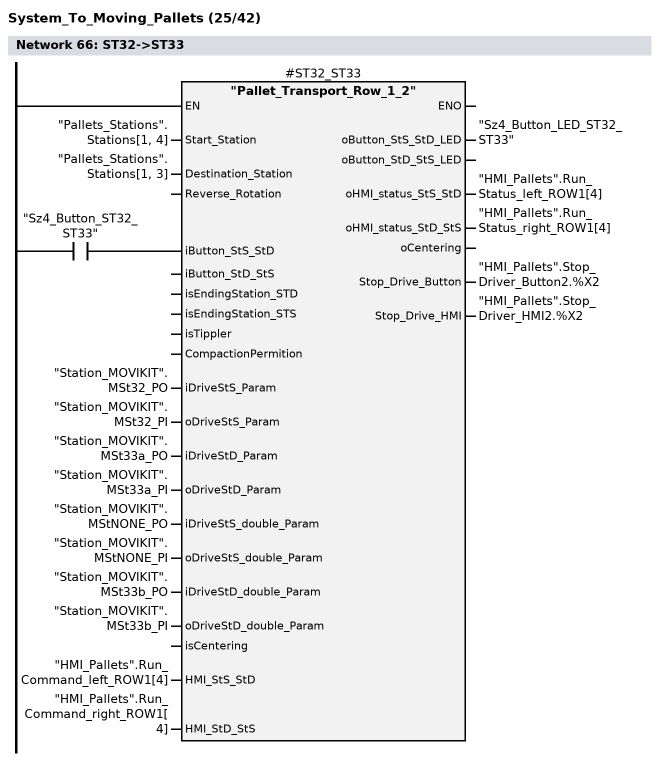
   RUNG wire#powerrail
      #ST32_ST33(iButton_StS_StD := wire#w1, Start_Station := "Pallets_Stations".Stations[1, 4], Destination_Station := "Pallets_Stations".Stations[1, 3], Reverse_Rotation :=, iButton_StD_StS :=, isEndingStation_STD :=, isEndingStation_STS :=, isTippler :=, CompactionPermition :=, iDriveStS_Param := "Station_MOVIKIT".MSt32_PO, oDriveStS_Param := "Station_MOVIKIT".MSt32_PI, iDriveStD_Param := "Station_MOVIKIT".MSt33a_PO, oDriveStD_Param := "Station_MOVIKIT".MSt33a_PI, iDriveStS_double_Param := "Station_MOVIKIT".MStNONE_PO, oDriveStS_double_Param := "Station_MOVIKIT".MStNONE_PI, iDriveStD_double_Param := "Station_MOVIKIT".MSt33b_PO, oDriveStD_double_Param := "Station_MOVIKIT".MSt33b_PI, isCentering :=, HMI_StS_StD := "HMI_Pallets".Run_Command_left_ROW1[4], HMI_StD_StS := "HMI_Pallets".Run_Command_right_ROW1[4], oButton_StS_StD_LED => "Sz4_Button_LED_ST32_ST33", oButton_StD_StS_LED =>, oHMI_status_StS_StD => "HMI_Pallets".Run_Status_left_ROW1[4], oHMI_status_StD_StS => "HMI_Pallets".Run_Status_right_ROW1[4], oCentering =>, Stop_Drive_Button => "HMI_Pallets".Stop_Driver_Button2.%X2, Stop_Drive_HMI => "HMI_Pallets".Stop_Driver_HMI2.%X2)
   END_RUNG
   RUNG wire#powerrail
      Contact( "Sz4_Button_ST32_ST33" )
   END_RUNG wire#w1
   // the same network as SCL:
   #ST32_ST33(Start_Station := "Pallets_Stations".Stations[1, 4],   // "Pallet_Transport_Row_1_2"
              Destination_Station := "Pallets_Stations".Stations[1, 3],
              iButton_StS_StD := "Sz4_Button_ST32_ST33",
              iDriveStS_Param := "Station_MOVIKIT".MSt32_PO,
              oDriveStS_Param := "Station_MOVIKIT".MSt32_PI,
              iDriveStD_Param := "Station_MOVIKIT".MSt33a_PO,
              oDriveStD_Param := "Station_MOVIKIT".MSt33a_PI,
              iDriveStS_double_Param := "Station_MOVIKIT".MStNONE_PO,
              oDriveStS_double_Param := "Station_MOVIKIT".MStNONE_PI,
              iDriveStD_double_Param := "Station_MOVIKIT".MSt33b_PO,
              oDriveStD_double_Param := "Station_MOVIKIT".MSt33b_PI,
              HMI_StS_StD := "HMI_Pallets".Run_Command_left_ROW1[4],
              HMI_StD_StS := "HMI_Pallets".Run_Command_right_ROW1[4],
              oButton_StS_StD_LED => "Sz4_Button_LED_ST32_ST33",
              oHMI_status_StS_StD => "HMI_Pallets".Run_Status_left_ROW1[4],
              oHMI_status_StD_StS => "HMI_Pallets".Run_Status_right_ROW1[4],
              Stop_Drive_Button => "HMI_Pallets".Stop_Driver_Button2.%X2,
              Stop_Drive_HMI => "HMI_Pallets".Stop_Driver_HMI2.%X2);
END_REGION

REGION Network 67: ST31->ST32
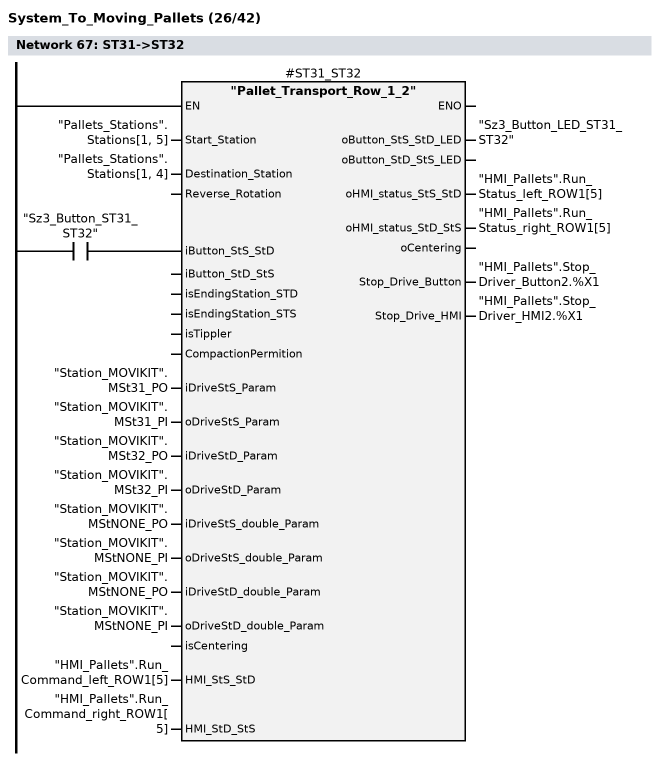
   RUNG wire#powerrail
      #ST31_ST32(iButton_StS_StD := wire#w1, Start_Station := "Pallets_Stations".Stations[1, 5], Destination_Station := "Pallets_Stations".Stations[1, 4], Reverse_Rotation :=, iButton_StD_StS :=, isEndingStation_STD :=, isEndingStation_STS :=, isTippler :=, CompactionPermition :=, iDriveStS_Param := "Station_MOVIKIT".MSt31_PO, oDriveStS_Param := "Station_MOVIKIT".MSt31_PI, iDriveStD_Param := "Station_MOVIKIT".MSt32_PO, oDriveStD_Param := "Station_MOVIKIT".MSt32_PI, iDriveStS_double_Param := "Station_MOVIKIT".MStNONE_PO, oDriveStS_double_Param := "Station_MOVIKIT".MStNONE_PI, iDriveStD_double_Param := "Station_MOVIKIT".MStNONE_PO, oDriveStD_double_Param := "Station_MOVIKIT".MStNONE_PI, isCentering :=, HMI_StS_StD := "HMI_Pallets".Run_Command_left_ROW1[5], HMI_StD_StS := "HMI_Pallets".Run_Command_right_ROW1[5], oButton_StS_StD_LED => "Sz3_Button_LED_ST31_ST32", oButton_StD_StS_LED =>, oHMI_status_StS_StD => "HMI_Pallets".Run_Status_left_ROW1[5], oHMI_status_StD_StS => "HMI_Pallets".Run_Status_right_ROW1[5], oCentering =>, Stop_Drive_Button => "HMI_Pallets".Stop_Driver_Button2.%X1, Stop_Drive_HMI => "HMI_Pallets".Stop_Driver_HMI2.%X1)
   END_RUNG
   RUNG wire#powerrail
      Contact( "Sz3_Button_ST31_ST32" )
   END_RUNG wire#w1
   // the same network as SCL:
   #ST31_ST32(Start_Station := "Pallets_Stations".Stations[1, 5],   // "Pallet_Transport_Row_1_2"
              Destination_Station := "Pallets_Stations".Stations[1, 4],
              iButton_StS_StD := "Sz3_Button_ST31_ST32",
              iDriveStS_Param := "Station_MOVIKIT".MSt31_PO,
              oDriveStS_Param := "Station_MOVIKIT".MSt31_PI,
              iDriveStD_Param := "Station_MOVIKIT".MSt32_PO,
              oDriveStD_Param := "Station_MOVIKIT".MSt32_PI,
              iDriveStS_double_Param := "Station_MOVIKIT".MStNONE_PO,
              oDriveStS_double_Param := "Station_MOVIKIT".MStNONE_PI,
              iDriveStD_double_Param := "Station_MOVIKIT".MStNONE_PO,
              oDriveStD_double_Param := "Station_MOVIKIT".MStNONE_PI,
              HMI_StS_StD := "HMI_Pallets".Run_Command_left_ROW1[5],
              HMI_StD_StS := "HMI_Pallets".Run_Command_right_ROW1[5],
              oButton_StS_StD_LED => "Sz3_Button_LED_ST31_ST32",
              oHMI_status_StS_StD => "HMI_Pallets".Run_Status_left_ROW1[5],
              oHMI_status_StD_StS => "HMI_Pallets".Run_Status_right_ROW1[5],
              Stop_Drive_Button => "HMI_Pallets".Stop_Driver_Button2.%X1,
              Stop_Drive_HMI => "HMI_Pallets".Stop_Driver_HMI2.%X1);
END_REGION

REGION Network 68: ST30->ST31
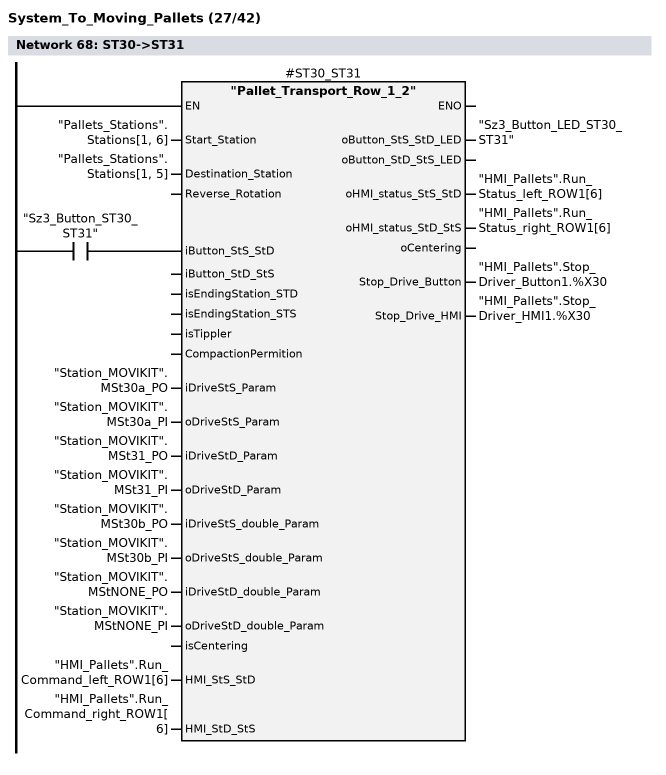
   RUNG wire#powerrail
      #ST30_ST31(iButton_StS_StD := wire#w1, Start_Station := "Pallets_Stations".Stations[1, 6], Destination_Station := "Pallets_Stations".Stations[1, 5], Reverse_Rotation :=, iButton_StD_StS :=, isEndingStation_STD :=, isEndingStation_STS :=, isTippler :=, CompactionPermition :=, iDriveStS_Param := "Station_MOVIKIT".MSt30a_PO, oDriveStS_Param := "Station_MOVIKIT".MSt30a_PI, iDriveStD_Param := "Station_MOVIKIT".MSt31_PO, oDriveStD_Param := "Station_MOVIKIT".MSt31_PI, iDriveStS_double_Param := "Station_MOVIKIT".MSt30b_PO, oDriveStS_double_Param := "Station_MOVIKIT".MSt30b_PI, iDriveStD_double_Param := "Station_MOVIKIT".MStNONE_PO, oDriveStD_double_Param := "Station_MOVIKIT".MStNONE_PI, isCentering :=, HMI_StS_StD := "HMI_Pallets".Run_Command_left_ROW1[6], HMI_StD_StS := "HMI_Pallets".Run_Command_right_ROW1[6], oButton_StS_StD_LED => "Sz3_Button_LED_ST30_ST31", oButton_StD_StS_LED =>, oHMI_status_StS_StD => "HMI_Pallets".Run_Status_left_ROW1[6], oHMI_status_StD_StS => "HMI_Pallets".Run_Status_right_ROW1[6], oCentering =>, Stop_Drive_Button => "HMI_Pallets".Stop_Driver_Button1.%X30, Stop_Drive_HMI => "HMI_Pallets".Stop_Driver_HMI1.%X30)
   END_RUNG
   RUNG wire#powerrail
      Contact( "Sz3_Button_ST30_ST31" )
   END_RUNG wire#w1
   // the same network as SCL:
   #ST30_ST31(Start_Station := "Pallets_Stations".Stations[1, 6],   // "Pallet_Transport_Row_1_2"
              Destination_Station := "Pallets_Stations".Stations[1, 5],
              iButton_StS_StD := "Sz3_Button_ST30_ST31",
              iDriveStS_Param := "Station_MOVIKIT".MSt30a_PO,
              oDriveStS_Param := "Station_MOVIKIT".MSt30a_PI,
              iDriveStD_Param := "Station_MOVIKIT".MSt31_PO,
              oDriveStD_Param := "Station_MOVIKIT".MSt31_PI,
              iDriveStS_double_Param := "Station_MOVIKIT".MSt30b_PO,
              oDriveStS_double_Param := "Station_MOVIKIT".MSt30b_PI,
              iDriveStD_double_Param := "Station_MOVIKIT".MStNONE_PO,
              oDriveStD_double_Param := "Station_MOVIKIT".MStNONE_PI,
              HMI_StS_StD := "HMI_Pallets".Run_Command_left_ROW1[6],
              HMI_StD_StS := "HMI_Pallets".Run_Command_right_ROW1[6],
              oButton_StS_StD_LED => "Sz3_Button_LED_ST30_ST31",
              oHMI_status_StS_StD => "HMI_Pallets".Run_Status_left_ROW1[6],
              oHMI_status_StD_StS => "HMI_Pallets".Run_Status_right_ROW1[6],
              Stop_Drive_Button => "HMI_Pallets".Stop_Driver_Button1.%X30,
              Stop_Drive_HMI => "HMI_Pallets".Stop_Driver_HMI1.%X30);
END_REGION

REGION Network 69: ST29->ST30
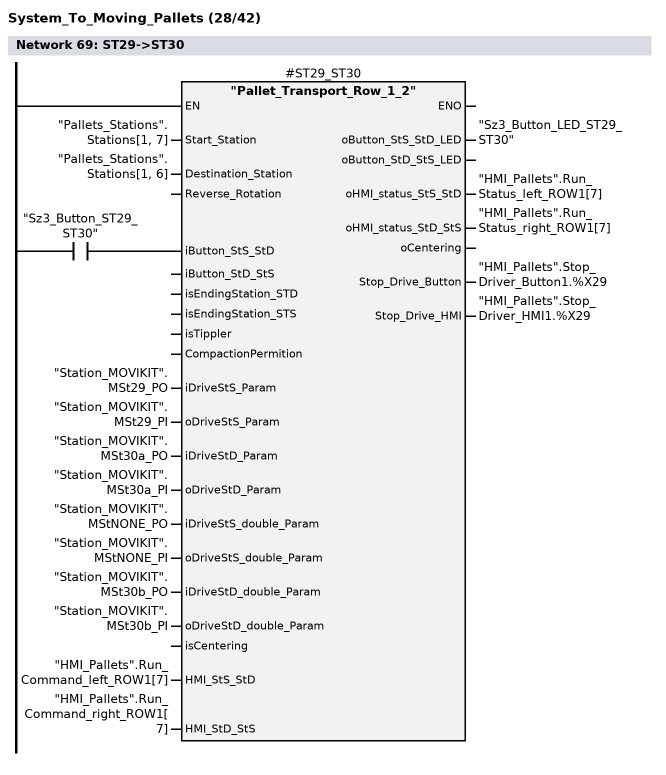
   RUNG wire#powerrail
      #ST29_ST30(iButton_StS_StD := wire#w1, Start_Station := "Pallets_Stations".Stations[1, 7], Destination_Station := "Pallets_Stations".Stations[1, 6], Reverse_Rotation :=, iButton_StD_StS :=, isEndingStation_STD :=, isEndingStation_STS :=, isTippler :=, CompactionPermition :=, iDriveStS_Param := "Station_MOVIKIT".MSt29_PO, oDriveStS_Param := "Station_MOVIKIT".MSt29_PI, iDriveStD_Param := "Station_MOVIKIT".MSt30a_PO, oDriveStD_Param := "Station_MOVIKIT".MSt30a_PI, iDriveStS_double_Param := "Station_MOVIKIT".MStNONE_PO, oDriveStS_double_Param := "Station_MOVIKIT".MStNONE_PI, iDriveStD_double_Param := "Station_MOVIKIT".MSt30b_PO, oDriveStD_double_Param := "Station_MOVIKIT".MSt30b_PI, isCentering :=, HMI_StS_StD := "HMI_Pallets".Run_Command_left_ROW1[7], HMI_StD_StS := "HMI_Pallets".Run_Command_right_ROW1[7], oButton_StS_StD_LED => "Sz3_Button_LED_ST29_ST30", oButton_StD_StS_LED =>, oHMI_status_StS_StD => "HMI_Pallets".Run_Status_left_ROW1[7], oHMI_status_StD_StS => "HMI_Pallets".Run_Status_right_ROW1[7], oCentering =>, Stop_Drive_Button => "HMI_Pallets".Stop_Driver_Button1.%X29, Stop_Drive_HMI => "HMI_Pallets".Stop_Driver_HMI1.%X29)
   END_RUNG
   RUNG wire#powerrail
      Contact( "Sz3_Button_ST29_ST30" )
   END_RUNG wire#w1
   // the same network as SCL:
   #ST29_ST30(Start_Station := "Pallets_Stations".Stations[1, 7],   // "Pallet_Transport_Row_1_2"
              Destination_Station := "Pallets_Stations".Stations[1, 6],
              iButton_StS_StD := "Sz3_Button_ST29_ST30",
              iDriveStS_Param := "Station_MOVIKIT".MSt29_PO,
              oDriveStS_Param := "Station_MOVIKIT".MSt29_PI,
              iDriveStD_Param := "Station_MOVIKIT".MSt30a_PO,
              oDriveStD_Param := "Station_MOVIKIT".MSt30a_PI,
              iDriveStS_double_Param := "Station_MOVIKIT".MStNONE_PO,
              oDriveStS_double_Param := "Station_MOVIKIT".MStNONE_PI,
              iDriveStD_double_Param := "Station_MOVIKIT".MSt30b_PO,
              oDriveStD_double_Param := "Station_MOVIKIT".MSt30b_PI,
              HMI_StS_StD := "HMI_Pallets".Run_Command_left_ROW1[7],
              HMI_StD_StS := "HMI_Pallets".Run_Command_right_ROW1[7],
              oButton_StS_StD_LED => "Sz3_Button_LED_ST29_ST30",
              oHMI_status_StS_StD => "HMI_Pallets".Run_Status_left_ROW1[7],
              oHMI_status_StD_StS => "HMI_Pallets".Run_Status_right_ROW1[7],
              Stop_Drive_Button => "HMI_Pallets".Stop_Driver_Button1.%X29,
              Stop_Drive_HMI => "HMI_Pallets".Stop_Driver_HMI1.%X29);
END_REGION

REGION Network 70: ST28->ST29
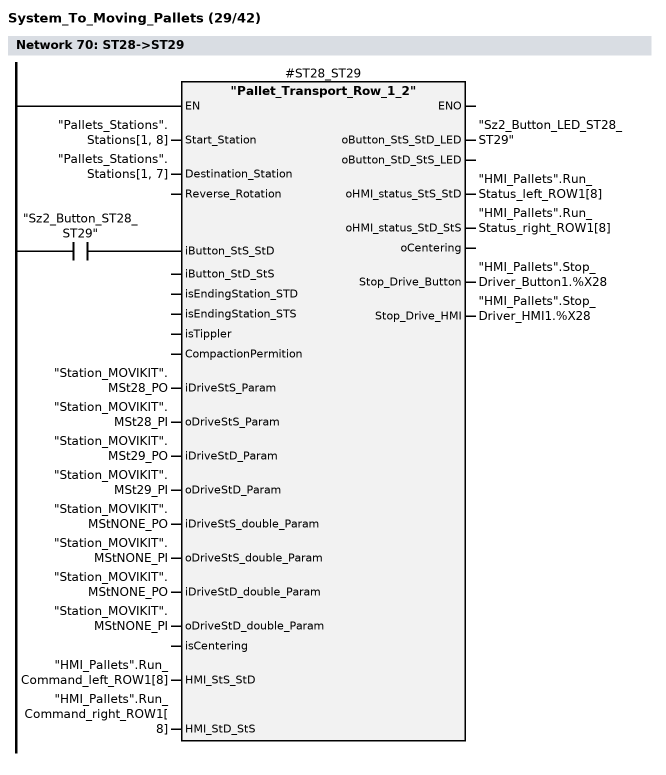
   RUNG wire#powerrail
      #ST28_ST29(iButton_StS_StD := wire#w1, Start_Station := "Pallets_Stations".Stations[1, 8], Destination_Station := "Pallets_Stations".Stations[1, 7], Reverse_Rotation :=, iButton_StD_StS :=, isEndingStation_STD :=, isEndingStation_STS :=, isTippler :=, CompactionPermition :=, iDriveStS_Param := "Station_MOVIKIT".MSt28_PO, oDriveStS_Param := "Station_MOVIKIT".MSt28_PI, iDriveStD_Param := "Station_MOVIKIT".MSt29_PO, oDriveStD_Param := "Station_MOVIKIT".MSt29_PI, iDriveStS_double_Param := "Station_MOVIKIT".MStNONE_PO, oDriveStS_double_Param := "Station_MOVIKIT".MStNONE_PI, iDriveStD_double_Param := "Station_MOVIKIT".MStNONE_PO, oDriveStD_double_Param := "Station_MOVIKIT".MStNONE_PI, isCentering :=, HMI_StS_StD := "HMI_Pallets".Run_Command_left_ROW1[8], HMI_StD_StS := "HMI_Pallets".Run_Command_right_ROW1[8], oButton_StS_StD_LED => "Sz2_Button_LED_ST28_ST29", oButton_StD_StS_LED =>, oHMI_status_StS_StD => "HMI_Pallets".Run_Status_left_ROW1[8], oHMI_status_StD_StS => "HMI_Pallets".Run_Status_right_ROW1[8], oCentering =>, Stop_Drive_Button => "HMI_Pallets".Stop_Driver_Button1.%X28, Stop_Drive_HMI => "HMI_Pallets".Stop_Driver_HMI1.%X28)
   END_RUNG
   RUNG wire#powerrail
      Contact( "Sz2_Button_ST28_ST29" )
   END_RUNG wire#w1
   // the same network as SCL:
   #ST28_ST29(Start_Station := "Pallets_Stations".Stations[1, 8],   // "Pallet_Transport_Row_1_2"
              Destination_Station := "Pallets_Stations".Stations[1, 7],
              iButton_StS_StD := "Sz2_Button_ST28_ST29",
              iDriveStS_Param := "Station_MOVIKIT".MSt28_PO,
              oDriveStS_Param := "Station_MOVIKIT".MSt28_PI,
              iDriveStD_Param := "Station_MOVIKIT".MSt29_PO,
              oDriveStD_Param := "Station_MOVIKIT".MSt29_PI,
              iDriveStS_double_Param := "Station_MOVIKIT".MStNONE_PO,
              oDriveStS_double_Param := "Station_MOVIKIT".MStNONE_PI,
              iDriveStD_double_Param := "Station_MOVIKIT".MStNONE_PO,
              oDriveStD_double_Param := "Station_MOVIKIT".MStNONE_PI,
              HMI_StS_StD := "HMI_Pallets".Run_Command_left_ROW1[8],
              HMI_StD_StS := "HMI_Pallets".Run_Command_right_ROW1[8],
              oButton_StS_StD_LED => "Sz2_Button_LED_ST28_ST29",
              oHMI_status_StS_StD => "HMI_Pallets".Run_Status_left_ROW1[8],
              oHMI_status_StD_StS => "HMI_Pallets".Run_Status_right_ROW1[8],
              Stop_Drive_Button => "HMI_Pallets".Stop_Driver_Button1.%X28,
              Stop_Drive_HMI => "HMI_Pallets".Stop_Driver_HMI1.%X28);
END_REGION

REGION Network 71: ST27->ST28
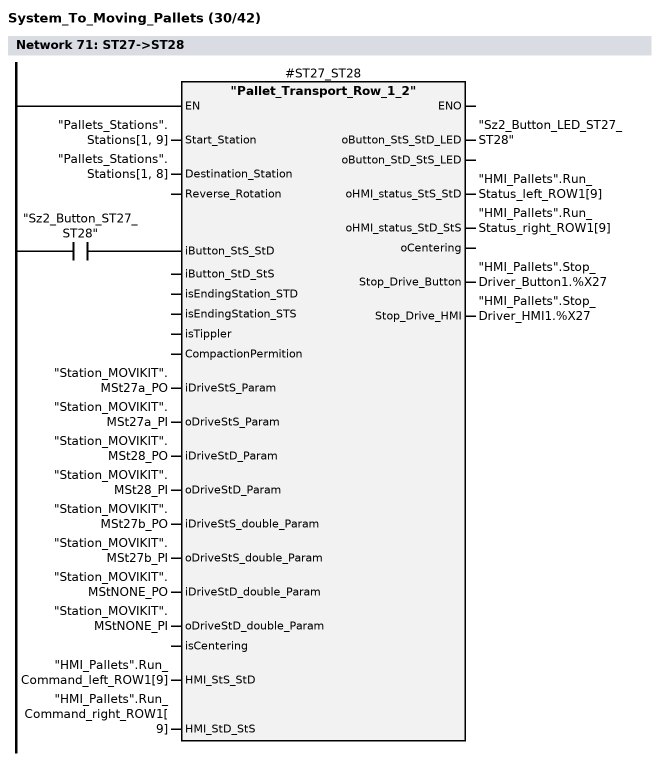
   RUNG wire#powerrail
      #ST27_ST28(iButton_StS_StD := wire#w1, Start_Station := "Pallets_Stations".Stations[1, 9], Destination_Station := "Pallets_Stations".Stations[1, 8], Reverse_Rotation :=, iButton_StD_StS :=, isEndingStation_STD :=, isEndingStation_STS :=, isTippler :=, CompactionPermition :=, iDriveStS_Param := "Station_MOVIKIT".MSt27a_PO, oDriveStS_Param := "Station_MOVIKIT".MSt27a_PI, iDriveStD_Param := "Station_MOVIKIT".MSt28_PO, oDriveStD_Param := "Station_MOVIKIT".MSt28_PI, iDriveStS_double_Param := "Station_MOVIKIT".MSt27b_PO, oDriveStS_double_Param := "Station_MOVIKIT".MSt27b_PI, iDriveStD_double_Param := "Station_MOVIKIT".MStNONE_PO, oDriveStD_double_Param := "Station_MOVIKIT".MStNONE_PI, isCentering :=, HMI_StS_StD := "HMI_Pallets".Run_Command_left_ROW1[9], HMI_StD_StS := "HMI_Pallets".Run_Command_right_ROW1[9], oButton_StS_StD_LED => "Sz2_Button_LED_ST27_ST28", oButton_StD_StS_LED =>, oHMI_status_StS_StD => "HMI_Pallets".Run_Status_left_ROW1[9], oHMI_status_StD_StS => "HMI_Pallets".Run_Status_right_ROW1[9], oCentering =>, Stop_Drive_Button => "HMI_Pallets".Stop_Driver_Button1.%X27, Stop_Drive_HMI => "HMI_Pallets".Stop_Driver_HMI1.%X27)
   END_RUNG
   RUNG wire#powerrail
      Contact( "Sz2_Button_ST27_ST28" )
   END_RUNG wire#w1
   // the same network as SCL:
   #ST27_ST28(Start_Station := "Pallets_Stations".Stations[1, 9],   // "Pallet_Transport_Row_1_2"
              Destination_Station := "Pallets_Stations".Stations[1, 8],
              iButton_StS_StD := "Sz2_Button_ST27_ST28",
              iDriveStS_Param := "Station_MOVIKIT".MSt27a_PO,
              oDriveStS_Param := "Station_MOVIKIT".MSt27a_PI,
              iDriveStD_Param := "Station_MOVIKIT".MSt28_PO,
              oDriveStD_Param := "Station_MOVIKIT".MSt28_PI,
              iDriveStS_double_Param := "Station_MOVIKIT".MSt27b_PO,
              oDriveStS_double_Param := "Station_MOVIKIT".MSt27b_PI,
              iDriveStD_double_Param := "Station_MOVIKIT".MStNONE_PO,
              oDriveStD_double_Param := "Station_MOVIKIT".MStNONE_PI,
              HMI_StS_StD := "HMI_Pallets".Run_Command_left_ROW1[9],
              HMI_StD_StS := "HMI_Pallets".Run_Command_right_ROW1[9],
              oButton_StS_StD_LED => "Sz2_Button_LED_ST27_ST28",
              oHMI_status_StS_StD => "HMI_Pallets".Run_Status_left_ROW1[9],
              oHMI_status_StD_StS => "HMI_Pallets".Run_Status_right_ROW1[9],
              Stop_Drive_Button => "HMI_Pallets".Stop_Driver_Button1.%X27,
              Stop_Drive_HMI => "HMI_Pallets".Stop_Driver_HMI1.%X27);
END_REGION

REGION Network 72: ST26->ST27
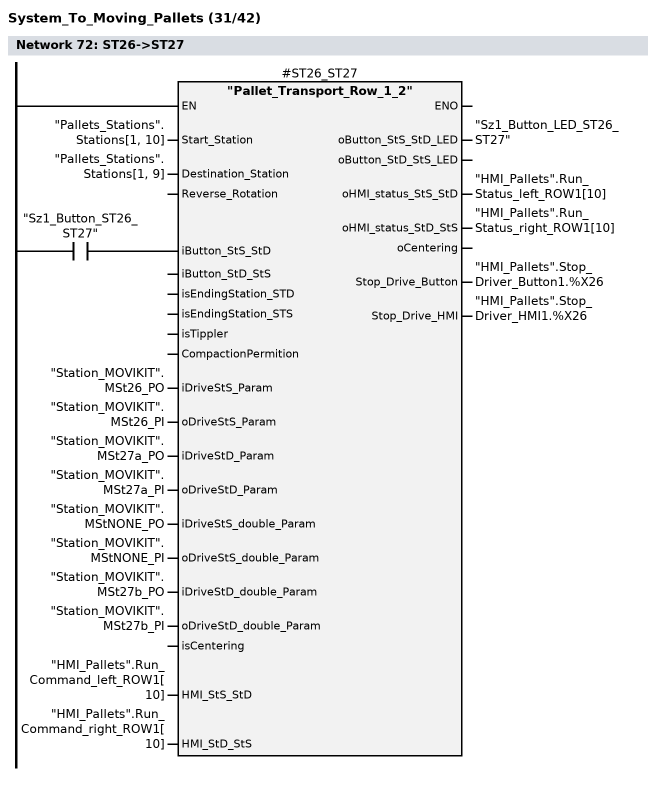
   RUNG wire#powerrail
      #ST26_ST27(iButton_StS_StD := wire#w1, Start_Station := "Pallets_Stations".Stations[1, 10], Destination_Station := "Pallets_Stations".Stations[1, 9], Reverse_Rotation :=, iButton_StD_StS :=, isEndingStation_STD :=, isEndingStation_STS :=, isTippler :=, CompactionPermition :=, iDriveStS_Param := "Station_MOVIKIT".MSt26_PO, oDriveStS_Param := "Station_MOVIKIT".MSt26_PI, iDriveStD_Param := "Station_MOVIKIT".MSt27a_PO, oDriveStD_Param := "Station_MOVIKIT".MSt27a_PI, iDriveStS_double_Param := "Station_MOVIKIT".MStNONE_PO, oDriveStS_double_Param := "Station_MOVIKIT".MStNONE_PI, iDriveStD_double_Param := "Station_MOVIKIT".MSt27b_PO, oDriveStD_double_Param := "Station_MOVIKIT".MSt27b_PI, isCentering :=, HMI_StS_StD := "HMI_Pallets".Run_Command_left_ROW1[10], HMI_StD_StS := "HMI_Pallets".Run_Command_right_ROW1[10], oButton_StS_StD_LED => "Sz1_Button_LED_ST26_ST27", oButton_StD_StS_LED =>, oHMI_status_StS_StD => "HMI_Pallets".Run_Status_left_ROW1[10], oHMI_status_StD_StS => "HMI_Pallets".Run_Status_right_ROW1[10], oCentering =>, Stop_Drive_Button => "HMI_Pallets".Stop_Driver_Button1.%X26, Stop_Drive_HMI => "HMI_Pallets".Stop_Driver_HMI1.%X26)
   END_RUNG
   RUNG wire#powerrail
      Contact( "Sz1_Button_ST26_ST27" )
   END_RUNG wire#w1
   // the same network as SCL:
   #ST26_ST27(Start_Station := "Pallets_Stations".Stations[1, 10],   // "Pallet_Transport_Row_1_2"
              Destination_Station := "Pallets_Stations".Stations[1, 9],
              iButton_StS_StD := "Sz1_Button_ST26_ST27",
              iDriveStS_Param := "Station_MOVIKIT".MSt26_PO,
              oDriveStS_Param := "Station_MOVIKIT".MSt26_PI,
              iDriveStD_Param := "Station_MOVIKIT".MSt27a_PO,
              oDriveStD_Param := "Station_MOVIKIT".MSt27a_PI,
              iDriveStS_double_Param := "Station_MOVIKIT".MStNONE_PO,
              oDriveStS_double_Param := "Station_MOVIKIT".MStNONE_PI,
              iDriveStD_double_Param := "Station_MOVIKIT".MSt27b_PO,
              oDriveStD_double_Param := "Station_MOVIKIT".MSt27b_PI,
              HMI_StS_StD := "HMI_Pallets".Run_Command_left_ROW1[10],
              HMI_StD_StS := "HMI_Pallets".Run_Command_right_ROW1[10],
              oButton_StS_StD_LED => "Sz1_Button_LED_ST26_ST27",
              oHMI_status_StS_StD => "HMI_Pallets".Run_Status_left_ROW1[10],
              oHMI_status_StD_StS => "HMI_Pallets".Run_Status_right_ROW1[10],
              Stop_Drive_Button => "HMI_Pallets".Stop_Driver_Button1.%X26,
              Stop_Drive_HMI => "HMI_Pallets".Stop_Driver_HMI1.%X26);
END_REGION

REGION Network 73: ST25->ST26
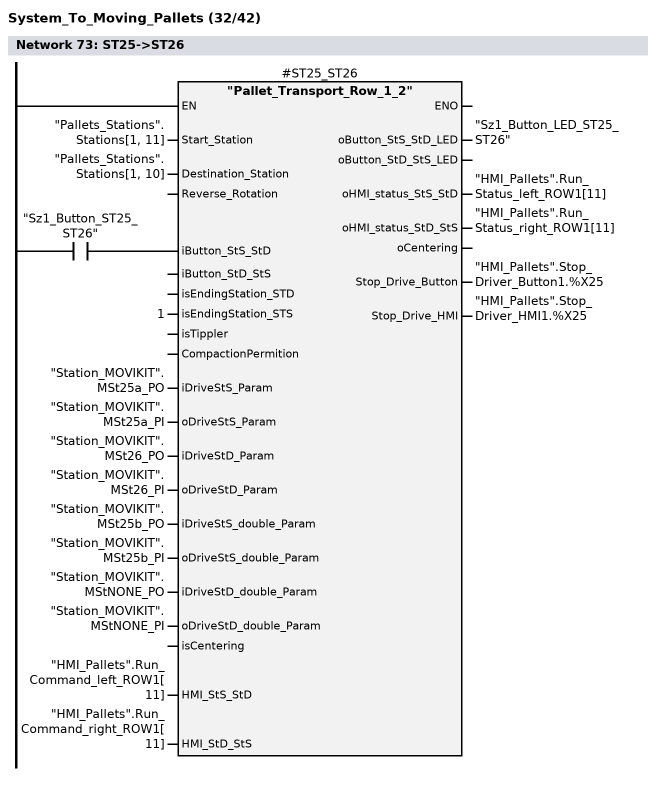
   RUNG wire#powerrail
      #ST25_ST26(iButton_StS_StD := wire#w1, Start_Station := "Pallets_Stations".Stations[1, 11], Destination_Station := "Pallets_Stations".Stations[1, 10], Reverse_Rotation :=, iButton_StD_StS :=, isEndingStation_STD :=, isEndingStation_STS := 1, isTippler :=, CompactionPermition :=, iDriveStS_Param := "Station_MOVIKIT".MSt25a_PO, oDriveStS_Param := "Station_MOVIKIT".MSt25a_PI, iDriveStD_Param := "Station_MOVIKIT".MSt26_PO, oDriveStD_Param := "Station_MOVIKIT".MSt26_PI, iDriveStS_double_Param := "Station_MOVIKIT".MSt25b_PO, oDriveStS_double_Param := "Station_MOVIKIT".MSt25b_PI, iDriveStD_double_Param := "Station_MOVIKIT".MStNONE_PO, oDriveStD_double_Param := "Station_MOVIKIT".MStNONE_PI, isCentering :=, HMI_StS_StD := "HMI_Pallets".Run_Command_left_ROW1[11], HMI_StD_StS := "HMI_Pallets".Run_Command_right_ROW1[11], oButton_StS_StD_LED => "Sz1_Button_LED_ST25_ST26", oButton_StD_StS_LED =>, oHMI_status_StS_StD => "HMI_Pallets".Run_Status_left_ROW1[11], oHMI_status_StD_StS => "HMI_Pallets".Run_Status_right_ROW1[11], oCentering =>, Stop_Drive_Button => "HMI_Pallets".Stop_Driver_Button1.%X25, Stop_Drive_HMI => "HMI_Pallets".Stop_Driver_HMI1.%X25)
   END_RUNG
   RUNG wire#powerrail
      Contact( "Sz1_Button_ST25_ST26" )
   END_RUNG wire#w1
   // the same network as SCL:
   #ST25_ST26(Start_Station := "Pallets_Stations".Stations[1, 11],   // "Pallet_Transport_Row_1_2"
              Destination_Station := "Pallets_Stations".Stations[1, 10],
              iButton_StS_StD := "Sz1_Button_ST25_ST26",
              isEndingStation_STS := 1,
              iDriveStS_Param := "Station_MOVIKIT".MSt25a_PO,
              oDriveStS_Param := "Station_MOVIKIT".MSt25a_PI,
              iDriveStD_Param := "Station_MOVIKIT".MSt26_PO,
              oDriveStD_Param := "Station_MOVIKIT".MSt26_PI,
              iDriveStS_double_Param := "Station_MOVIKIT".MSt25b_PO,
              oDriveStS_double_Param := "Station_MOVIKIT".MSt25b_PI,
              iDriveStD_double_Param := "Station_MOVIKIT".MStNONE_PO,
              oDriveStD_double_Param := "Station_MOVIKIT".MStNONE_PI,
              HMI_StS_StD := "HMI_Pallets".Run_Command_left_ROW1[11],
              HMI_StD_StS := "HMI_Pallets".Run_Command_right_ROW1[11],
              oButton_StS_StD_LED => "Sz1_Button_LED_ST25_ST26",
              oHMI_status_StS_StD => "HMI_Pallets".Run_Status_left_ROW1[11],
              oHMI_status_StD_StS => "HMI_Pallets".Run_Status_right_ROW1[11],
              Stop_Drive_Button => "HMI_Pallets".Stop_Driver_Button1.%X25,
              Stop_Drive_HMI => "HMI_Pallets".Stop_Driver_HMI1.%X25);
END_REGION

REGION Network 74: ST36->ST38
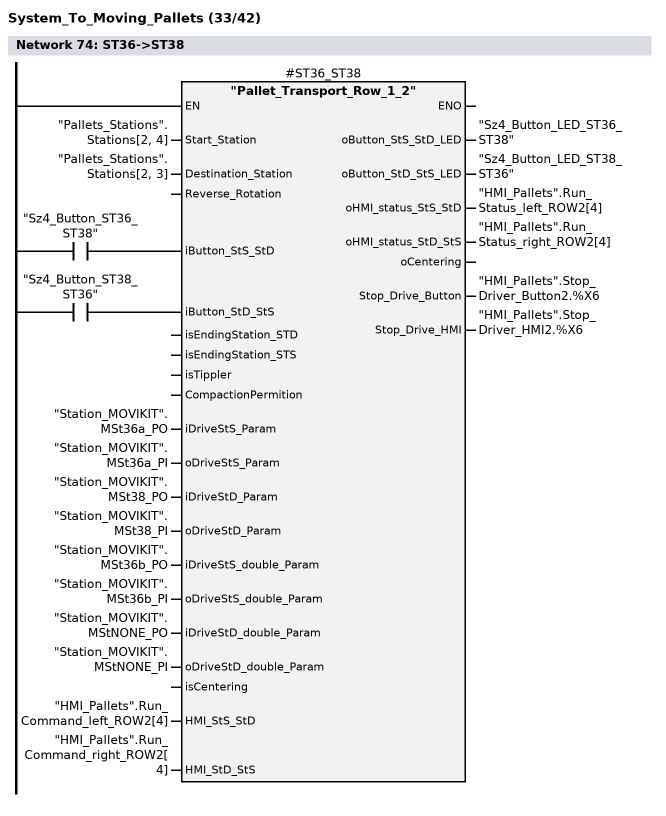
   RUNG wire#powerrail
      #ST36_ST38(iButton_StS_StD := wire#w1, iButton_StD_StS := wire#w2, Start_Station := "Pallets_Stations".Stations[2, 4], Destination_Station := "Pallets_Stations".Stations[2, 3], Reverse_Rotation :=, isEndingStation_STD :=, isEndingStation_STS :=, isTippler :=, CompactionPermition :=, iDriveStS_Param := "Station_MOVIKIT".MSt36a_PO, oDriveStS_Param := "Station_MOVIKIT".MSt36a_PI, iDriveStD_Param := "Station_MOVIKIT".MSt38_PO, oDriveStD_Param := "Station_MOVIKIT".MSt38_PI, iDriveStS_double_Param := "Station_MOVIKIT".MSt36b_PO, oDriveStS_double_Param := "Station_MOVIKIT".MSt36b_PI, iDriveStD_double_Param := "Station_MOVIKIT".MStNONE_PO, oDriveStD_double_Param := "Station_MOVIKIT".MStNONE_PI, isCentering :=, HMI_StS_StD := "HMI_Pallets".Run_Command_left_ROW2[4], HMI_StD_StS := "HMI_Pallets".Run_Command_right_ROW2[4], oButton_StS_StD_LED => "Sz4_Button_LED_ST36_ST38", oButton_StD_StS_LED => "Sz4_Button_LED_ST38_ST36", oHMI_status_StS_StD => "HMI_Pallets".Run_Status_left_ROW2[4], oHMI_status_StD_StS => "HMI_Pallets".Run_Status_right_ROW2[4], oCentering =>, Stop_Drive_Button => "HMI_Pallets".Stop_Driver_Button2.%X6, Stop_Drive_HMI => "HMI_Pallets".Stop_Driver_HMI2.%X6)
   END_RUNG
   RUNG wire#powerrail
      Contact( "Sz4_Button_ST36_ST38" )
   END_RUNG wire#w1
   RUNG wire#powerrail
      Contact( "Sz4_Button_ST38_ST36" )
   END_RUNG wire#w2
   // the same network as SCL:
   #ST36_ST38(Start_Station := "Pallets_Stations".Stations[2, 4],   // "Pallet_Transport_Row_1_2"
              Destination_Station := "Pallets_Stations".Stations[2, 3],
              iButton_StS_StD := "Sz4_Button_ST36_ST38",
              iButton_StD_StS := "Sz4_Button_ST38_ST36",
              iDriveStS_Param := "Station_MOVIKIT".MSt36a_PO,
              oDriveStS_Param := "Station_MOVIKIT".MSt36a_PI,
              iDriveStD_Param := "Station_MOVIKIT".MSt38_PO,
              oDriveStD_Param := "Station_MOVIKIT".MSt38_PI,
              iDriveStS_double_Param := "Station_MOVIKIT".MSt36b_PO,
              oDriveStS_double_Param := "Station_MOVIKIT".MSt36b_PI,
              iDriveStD_double_Param := "Station_MOVIKIT".MStNONE_PO,
              oDriveStD_double_Param := "Station_MOVIKIT".MStNONE_PI,
              HMI_StS_StD := "HMI_Pallets".Run_Command_left_ROW2[4],
              HMI_StD_StS := "HMI_Pallets".Run_Command_right_ROW2[4],
              oButton_StS_StD_LED => "Sz4_Button_LED_ST36_ST38",
              oButton_StD_StS_LED => "Sz4_Button_LED_ST38_ST36",
              oHMI_status_StS_StD => "HMI_Pallets".Run_Status_left_ROW2[4],
              oHMI_status_StD_StS => "HMI_Pallets".Run_Status_right_ROW2[4],
              Stop_Drive_Button => "HMI_Pallets".Stop_Driver_Button2.%X6,
              Stop_Drive_HMI => "HMI_Pallets".Stop_Driver_HMI2.%X6);
END_REGION

REGION Network 75: ST37->ST36
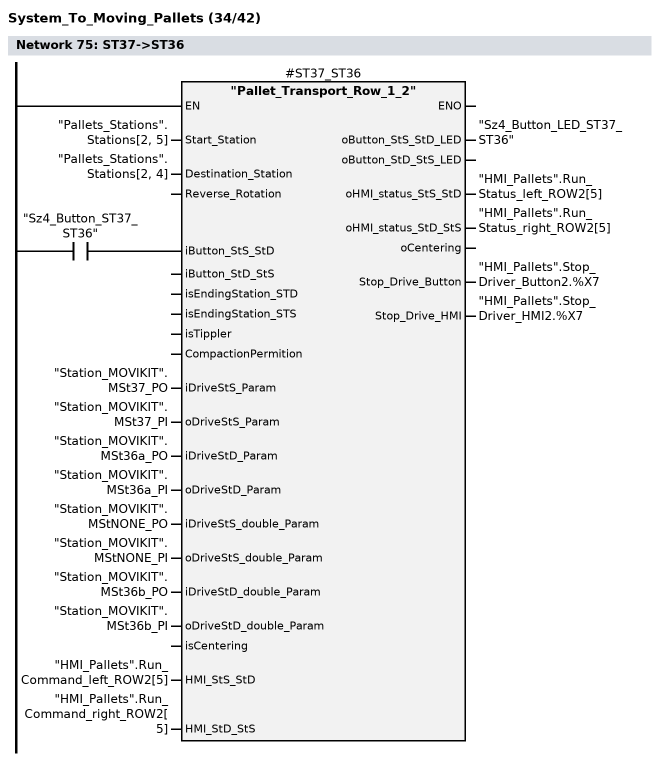
   RUNG wire#powerrail
      #ST37_ST36(iButton_StS_StD := wire#w1, Start_Station := "Pallets_Stations".Stations[2, 5], Destination_Station := "Pallets_Stations".Stations[2, 4], Reverse_Rotation :=, iButton_StD_StS :=, isEndingStation_STD :=, isEndingStation_STS :=, isTippler :=, CompactionPermition :=, iDriveStS_Param := "Station_MOVIKIT".MSt37_PO, oDriveStS_Param := "Station_MOVIKIT".MSt37_PI, iDriveStD_Param := "Station_MOVIKIT".MSt36a_PO, oDriveStD_Param := "Station_MOVIKIT".MSt36a_PI, iDriveStS_double_Param := "Station_MOVIKIT".MStNONE_PO, oDriveStS_double_Param := "Station_MOVIKIT".MStNONE_PI, iDriveStD_double_Param := "Station_MOVIKIT".MSt36b_PO, oDriveStD_double_Param := "Station_MOVIKIT".MSt36b_PI, isCentering :=, HMI_StS_StD := "HMI_Pallets".Run_Command_left_ROW2[5], HMI_StD_StS := "HMI_Pallets".Run_Command_right_ROW2[5], oButton_StS_StD_LED => "Sz4_Button_LED_ST37_ST36", oButton_StD_StS_LED =>, oHMI_status_StS_StD => "HMI_Pallets".Run_Status_left_ROW2[5], oHMI_status_StD_StS => "HMI_Pallets".Run_Status_right_ROW2[5], oCentering =>, Stop_Drive_Button => "HMI_Pallets".Stop_Driver_Button2.%X7, Stop_Drive_HMI => "HMI_Pallets".Stop_Driver_HMI2.%X7)
   END_RUNG
   RUNG wire#powerrail
      Contact( "Sz4_Button_ST37_ST36" )
   END_RUNG wire#w1
   // the same network as SCL:
   #ST37_ST36(Start_Station := "Pallets_Stations".Stations[2, 5],   // "Pallet_Transport_Row_1_2"
              Destination_Station := "Pallets_Stations".Stations[2, 4],
              iButton_StS_StD := "Sz4_Button_ST37_ST36",
              iDriveStS_Param := "Station_MOVIKIT".MSt37_PO,
              oDriveStS_Param := "Station_MOVIKIT".MSt37_PI,
              iDriveStD_Param := "Station_MOVIKIT".MSt36a_PO,
              oDriveStD_Param := "Station_MOVIKIT".MSt36a_PI,
              iDriveStS_double_Param := "Station_MOVIKIT".MStNONE_PO,
              oDriveStS_double_Param := "Station_MOVIKIT".MStNONE_PI,
              iDriveStD_double_Param := "Station_MOVIKIT".MSt36b_PO,
              oDriveStD_double_Param := "Station_MOVIKIT".MSt36b_PI,
              HMI_StS_StD := "HMI_Pallets".Run_Command_left_ROW2[5],
              HMI_StD_StS := "HMI_Pallets".Run_Command_right_ROW2[5],
              oButton_StS_StD_LED => "Sz4_Button_LED_ST37_ST36",
              oHMI_status_StS_StD => "HMI_Pallets".Run_Status_left_ROW2[5],
              oHMI_status_StD_StS => "HMI_Pallets".Run_Status_right_ROW2[5],
              Stop_Drive_Button => "HMI_Pallets".Stop_Driver_Button2.%X7,
              Stop_Drive_HMI => "HMI_Pallets".Stop_Driver_HMI2.%X7);
END_REGION

REGION Network 76: ST18->ST37
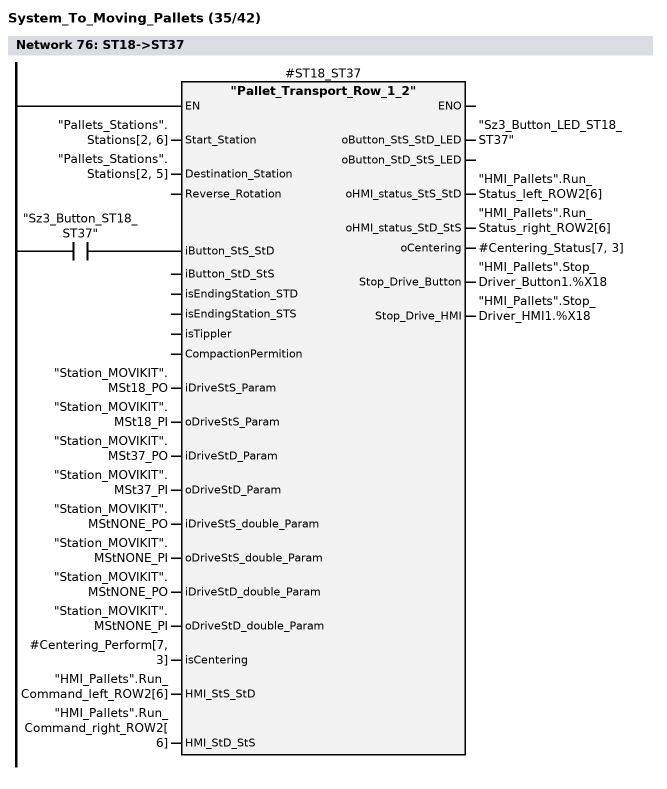
   RUNG wire#powerrail
      #ST18_ST37(iButton_StS_StD := wire#w1, Start_Station := "Pallets_Stations".Stations[2, 6], Destination_Station := "Pallets_Stations".Stations[2, 5], Reverse_Rotation :=, iButton_StD_StS :=, isEndingStation_STD :=, isEndingStation_STS :=, isTippler :=, CompactionPermition :=, iDriveStS_Param := "Station_MOVIKIT".MSt18_PO, oDriveStS_Param := "Station_MOVIKIT".MSt18_PI, iDriveStD_Param := "Station_MOVIKIT".MSt37_PO, oDriveStD_Param := "Station_MOVIKIT".MSt37_PI, iDriveStS_double_Param := "Station_MOVIKIT".MStNONE_PO, oDriveStS_double_Param := "Station_MOVIKIT".MStNONE_PI, iDriveStD_double_Param := "Station_MOVIKIT".MStNONE_PO, oDriveStD_double_Param := "Station_MOVIKIT".MStNONE_PI, isCentering := #Centering_Perform[7, 3], HMI_StS_StD := "HMI_Pallets".Run_Command_left_ROW2[6], HMI_StD_StS := "HMI_Pallets".Run_Command_right_ROW2[6], oButton_StS_StD_LED => "Sz3_Button_LED_ST18_ST37", oButton_StD_StS_LED =>, oHMI_status_StS_StD => "HMI_Pallets".Run_Status_left_ROW2[6], oHMI_status_StD_StS => "HMI_Pallets".Run_Status_right_ROW2[6], oCentering => #Centering_Status[7, 3], Stop_Drive_Button => "HMI_Pallets".Stop_Driver_Button1.%X18, Stop_Drive_HMI => "HMI_Pallets".Stop_Driver_HMI1.%X18)
   END_RUNG
   RUNG wire#powerrail
      Contact( "Sz3_Button_ST18_ST37" )
   END_RUNG wire#w1
   // the same network as SCL:
   #ST18_ST37(Start_Station := "Pallets_Stations".Stations[2, 6],   // "Pallet_Transport_Row_1_2"
              Destination_Station := "Pallets_Stations".Stations[2, 5],
              iButton_StS_StD := "Sz3_Button_ST18_ST37",
              iDriveStS_Param := "Station_MOVIKIT".MSt18_PO,
              oDriveStS_Param := "Station_MOVIKIT".MSt18_PI,
              iDriveStD_Param := "Station_MOVIKIT".MSt37_PO,
              oDriveStD_Param := "Station_MOVIKIT".MSt37_PI,
              iDriveStS_double_Param := "Station_MOVIKIT".MStNONE_PO,
              oDriveStS_double_Param := "Station_MOVIKIT".MStNONE_PI,
              iDriveStD_double_Param := "Station_MOVIKIT".MStNONE_PO,
              oDriveStD_double_Param := "Station_MOVIKIT".MStNONE_PI,
              isCentering := #Centering_Perform[7, 3],
              HMI_StS_StD := "HMI_Pallets".Run_Command_left_ROW2[6],
              HMI_StD_StS := "HMI_Pallets".Run_Command_right_ROW2[6],
              oButton_StS_StD_LED => "Sz3_Button_LED_ST18_ST37",
              oHMI_status_StS_StD => "HMI_Pallets".Run_Status_left_ROW2[6],
              oHMI_status_StD_StS => "HMI_Pallets".Run_Status_right_ROW2[6],
              oCentering => #Centering_Status[7, 3],
              Stop_Drive_Button => "HMI_Pallets".Stop_Driver_Button1.%X18,
              Stop_Drive_HMI => "HMI_Pallets".Stop_Driver_HMI1.%X18);
END_REGION

REGION Network 77: ST19->ST18
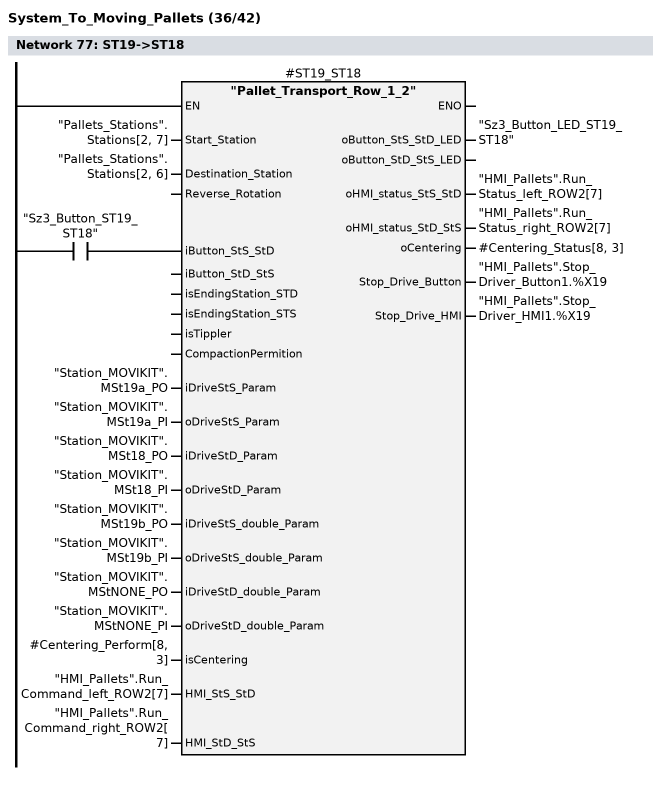
   RUNG wire#powerrail
      #ST19_ST18(iButton_StS_StD := wire#w1, Start_Station := "Pallets_Stations".Stations[2, 7], Destination_Station := "Pallets_Stations".Stations[2, 6], Reverse_Rotation :=, iButton_StD_StS :=, isEndingStation_STD :=, isEndingStation_STS :=, isTippler :=, CompactionPermition :=, iDriveStS_Param := "Station_MOVIKIT".MSt19a_PO, oDriveStS_Param := "Station_MOVIKIT".MSt19a_PI, iDriveStD_Param := "Station_MOVIKIT".MSt18_PO, oDriveStD_Param := "Station_MOVIKIT".MSt18_PI, iDriveStS_double_Param := "Station_MOVIKIT".MSt19b_PO, oDriveStS_double_Param := "Station_MOVIKIT".MSt19b_PI, iDriveStD_double_Param := "Station_MOVIKIT".MStNONE_PO, oDriveStD_double_Param := "Station_MOVIKIT".MStNONE_PI, isCentering := #Centering_Perform[8, 3], HMI_StS_StD := "HMI_Pallets".Run_Command_left_ROW2[7], HMI_StD_StS := "HMI_Pallets".Run_Command_right_ROW2[7], oButton_StS_StD_LED => "Sz3_Button_LED_ST19_ST18", oButton_StD_StS_LED =>, oHMI_status_StS_StD => "HMI_Pallets".Run_Status_left_ROW2[7], oHMI_status_StD_StS => "HMI_Pallets".Run_Status_right_ROW2[7], oCentering => #Centering_Status[8, 3], Stop_Drive_Button => "HMI_Pallets".Stop_Driver_Button1.%X19, Stop_Drive_HMI => "HMI_Pallets".Stop_Driver_HMI1.%X19)
   END_RUNG
   RUNG wire#powerrail
      Contact( "Sz3_Button_ST19_ST18" )
   END_RUNG wire#w1
   // the same network as SCL:
   #ST19_ST18(Start_Station := "Pallets_Stations".Stations[2, 7],   // "Pallet_Transport_Row_1_2"
              Destination_Station := "Pallets_Stations".Stations[2, 6],
              iButton_StS_StD := "Sz3_Button_ST19_ST18",
              iDriveStS_Param := "Station_MOVIKIT".MSt19a_PO,
              oDriveStS_Param := "Station_MOVIKIT".MSt19a_PI,
              iDriveStD_Param := "Station_MOVIKIT".MSt18_PO,
              oDriveStD_Param := "Station_MOVIKIT".MSt18_PI,
              iDriveStS_double_Param := "Station_MOVIKIT".MSt19b_PO,
              oDriveStS_double_Param := "Station_MOVIKIT".MSt19b_PI,
              iDriveStD_double_Param := "Station_MOVIKIT".MStNONE_PO,
              oDriveStD_double_Param := "Station_MOVIKIT".MStNONE_PI,
              isCentering := #Centering_Perform[8, 3],
              HMI_StS_StD := "HMI_Pallets".Run_Command_left_ROW2[7],
              HMI_StD_StS := "HMI_Pallets".Run_Command_right_ROW2[7],
              oButton_StS_StD_LED => "Sz3_Button_LED_ST19_ST18",
              oHMI_status_StS_StD => "HMI_Pallets".Run_Status_left_ROW2[7],
              oHMI_status_StD_StS => "HMI_Pallets".Run_Status_right_ROW2[7],
              oCentering => #Centering_Status[8, 3],
              Stop_Drive_Button => "HMI_Pallets".Stop_Driver_Button1.%X19,
              Stop_Drive_HMI => "HMI_Pallets".Stop_Driver_HMI1.%X19);
END_REGION

REGION Network 78: ST20->ST19
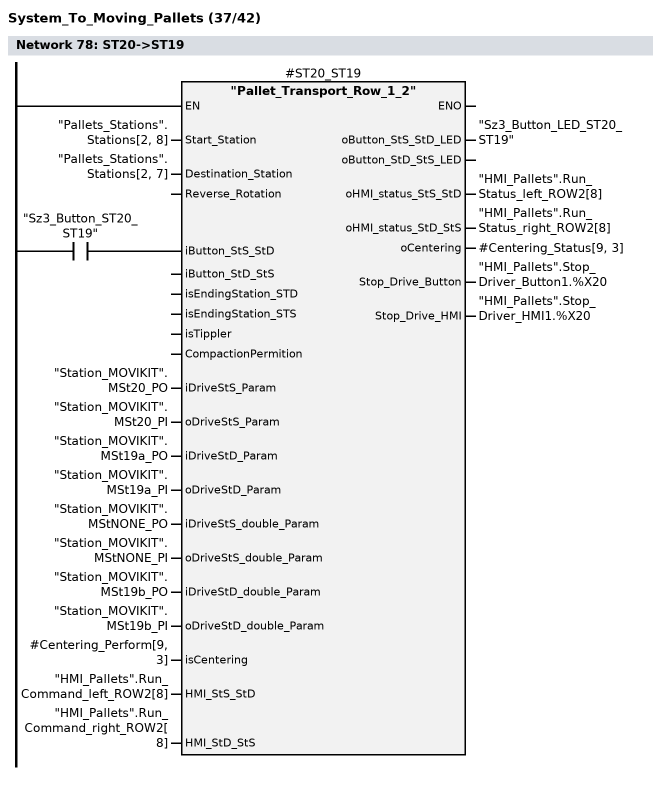
   RUNG wire#powerrail
      #ST20_ST19(iButton_StS_StD := wire#w1, Start_Station := "Pallets_Stations".Stations[2, 8], Destination_Station := "Pallets_Stations".Stations[2, 7], Reverse_Rotation :=, iButton_StD_StS :=, isEndingStation_STD :=, isEndingStation_STS :=, isTippler :=, CompactionPermition :=, iDriveStS_Param := "Station_MOVIKIT".MSt20_PO, oDriveStS_Param := "Station_MOVIKIT".MSt20_PI, iDriveStD_Param := "Station_MOVIKIT".MSt19a_PO, oDriveStD_Param := "Station_MOVIKIT".MSt19a_PI, iDriveStS_double_Param := "Station_MOVIKIT".MStNONE_PO, oDriveStS_double_Param := "Station_MOVIKIT".MStNONE_PI, iDriveStD_double_Param := "Station_MOVIKIT".MSt19b_PO, oDriveStD_double_Param := "Station_MOVIKIT".MSt19b_PI, isCentering := #Centering_Perform[9, 3], HMI_StS_StD := "HMI_Pallets".Run_Command_left_ROW2[8], HMI_StD_StS := "HMI_Pallets".Run_Command_right_ROW2[8], oButton_StS_StD_LED => "Sz3_Button_LED_ST20_ST19", oButton_StD_StS_LED =>, oHMI_status_StS_StD => "HMI_Pallets".Run_Status_left_ROW2[8], oHMI_status_StD_StS => "HMI_Pallets".Run_Status_right_ROW2[8], oCentering => #Centering_Status[9, 3], Stop_Drive_Button => "HMI_Pallets".Stop_Driver_Button1.%X20, Stop_Drive_HMI => "HMI_Pallets".Stop_Driver_HMI1.%X20)
   END_RUNG
   RUNG wire#powerrail
      Contact( "Sz3_Button_ST20_ST19" )
   END_RUNG wire#w1
   // the same network as SCL:
   #ST20_ST19(Start_Station := "Pallets_Stations".Stations[2, 8],   // "Pallet_Transport_Row_1_2"
              Destination_Station := "Pallets_Stations".Stations[2, 7],
              iButton_StS_StD := "Sz3_Button_ST20_ST19",
              iDriveStS_Param := "Station_MOVIKIT".MSt20_PO,
              oDriveStS_Param := "Station_MOVIKIT".MSt20_PI,
              iDriveStD_Param := "Station_MOVIKIT".MSt19a_PO,
              oDriveStD_Param := "Station_MOVIKIT".MSt19a_PI,
              iDriveStS_double_Param := "Station_MOVIKIT".MStNONE_PO,
              oDriveStS_double_Param := "Station_MOVIKIT".MStNONE_PI,
              iDriveStD_double_Param := "Station_MOVIKIT".MSt19b_PO,
              oDriveStD_double_Param := "Station_MOVIKIT".MSt19b_PI,
              isCentering := #Centering_Perform[9, 3],
              HMI_StS_StD := "HMI_Pallets".Run_Command_left_ROW2[8],
              HMI_StD_StS := "HMI_Pallets".Run_Command_right_ROW2[8],
              oButton_StS_StD_LED => "Sz3_Button_LED_ST20_ST19",
              oHMI_status_StS_StD => "HMI_Pallets".Run_Status_left_ROW2[8],
              oHMI_status_StD_StS => "HMI_Pallets".Run_Status_right_ROW2[8],
              oCentering => #Centering_Status[9, 3],
              Stop_Drive_Button => "HMI_Pallets".Stop_Driver_Button1.%X20,
              Stop_Drive_HMI => "HMI_Pallets".Stop_Driver_HMI1.%X20);
END_REGION

REGION Network 79: ST21->ST20
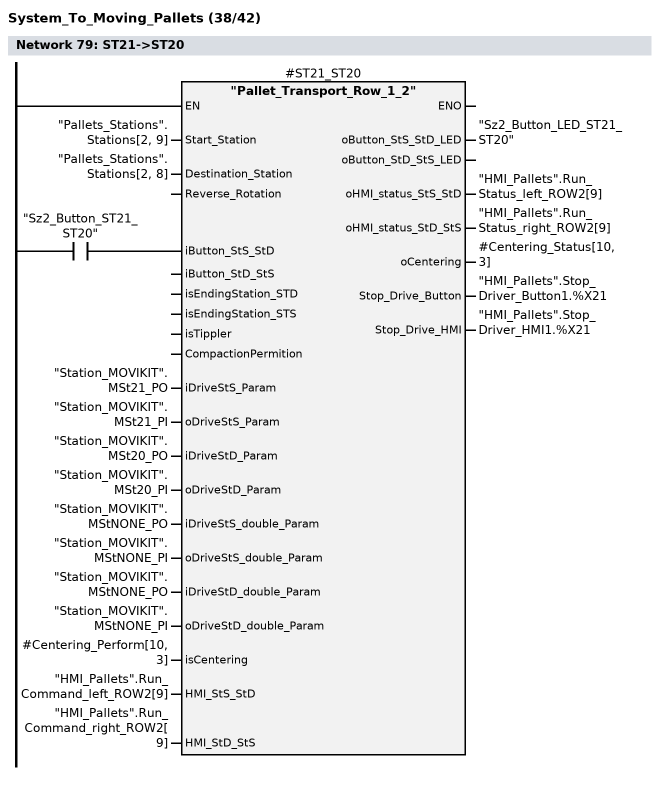
   RUNG wire#powerrail
      #ST21_ST20(iButton_StS_StD := wire#w1, Start_Station := "Pallets_Stations".Stations[2, 9], Destination_Station := "Pallets_Stations".Stations[2, 8], Reverse_Rotation :=, iButton_StD_StS :=, isEndingStation_STD :=, isEndingStation_STS :=, isTippler :=, CompactionPermition :=, iDriveStS_Param := "Station_MOVIKIT".MSt21_PO, oDriveStS_Param := "Station_MOVIKIT".MSt21_PI, iDriveStD_Param := "Station_MOVIKIT".MSt20_PO, oDriveStD_Param := "Station_MOVIKIT".MSt20_PI, iDriveStS_double_Param := "Station_MOVIKIT".MStNONE_PO, oDriveStS_double_Param := "Station_MOVIKIT".MStNONE_PI, iDriveStD_double_Param := "Station_MOVIKIT".MStNONE_PO, oDriveStD_double_Param := "Station_MOVIKIT".MStNONE_PI, isCentering := #Centering_Perform[10, 3], HMI_StS_StD := "HMI_Pallets".Run_Command_left_ROW2[9], HMI_StD_StS := "HMI_Pallets".Run_Command_right_ROW2[9], oButton_StS_StD_LED => "Sz2_Button_LED_ST21_ST20", oButton_StD_StS_LED =>, oHMI_status_StS_StD => "HMI_Pallets".Run_Status_left_ROW2[9], oHMI_status_StD_StS => "HMI_Pallets".Run_Status_right_ROW2[9], oCentering => #Centering_Status[10, 3], Stop_Drive_Button => "HMI_Pallets".Stop_Driver_Button1.%X21, Stop_Drive_HMI => "HMI_Pallets".Stop_Driver_HMI1.%X21)
   END_RUNG
   RUNG wire#powerrail
      Contact( "Sz2_Button_ST21_ST20" )
   END_RUNG wire#w1
   // the same network as SCL:
   #ST21_ST20(Start_Station := "Pallets_Stations".Stations[2, 9],   // "Pallet_Transport_Row_1_2"
              Destination_Station := "Pallets_Stations".Stations[2, 8],
              iButton_StS_StD := "Sz2_Button_ST21_ST20",
              iDriveStS_Param := "Station_MOVIKIT".MSt21_PO,
              oDriveStS_Param := "Station_MOVIKIT".MSt21_PI,
              iDriveStD_Param := "Station_MOVIKIT".MSt20_PO,
              oDriveStD_Param := "Station_MOVIKIT".MSt20_PI,
              iDriveStS_double_Param := "Station_MOVIKIT".MStNONE_PO,
              oDriveStS_double_Param := "Station_MOVIKIT".MStNONE_PI,
              iDriveStD_double_Param := "Station_MOVIKIT".MStNONE_PO,
              oDriveStD_double_Param := "Station_MOVIKIT".MStNONE_PI,
              isCentering := #Centering_Perform[10, 3],
              HMI_StS_StD := "HMI_Pallets".Run_Command_left_ROW2[9],
              HMI_StD_StS := "HMI_Pallets".Run_Command_right_ROW2[9],
              oButton_StS_StD_LED => "Sz2_Button_LED_ST21_ST20",
              oHMI_status_StS_StD => "HMI_Pallets".Run_Status_left_ROW2[9],
              oHMI_status_StD_StS => "HMI_Pallets".Run_Status_right_ROW2[9],
              oCentering => #Centering_Status[10, 3],
              Stop_Drive_Button => "HMI_Pallets".Stop_Driver_Button1.%X21,
              Stop_Drive_HMI => "HMI_Pallets".Stop_Driver_HMI1.%X21);
END_REGION

REGION Network 80: ST22->ST21
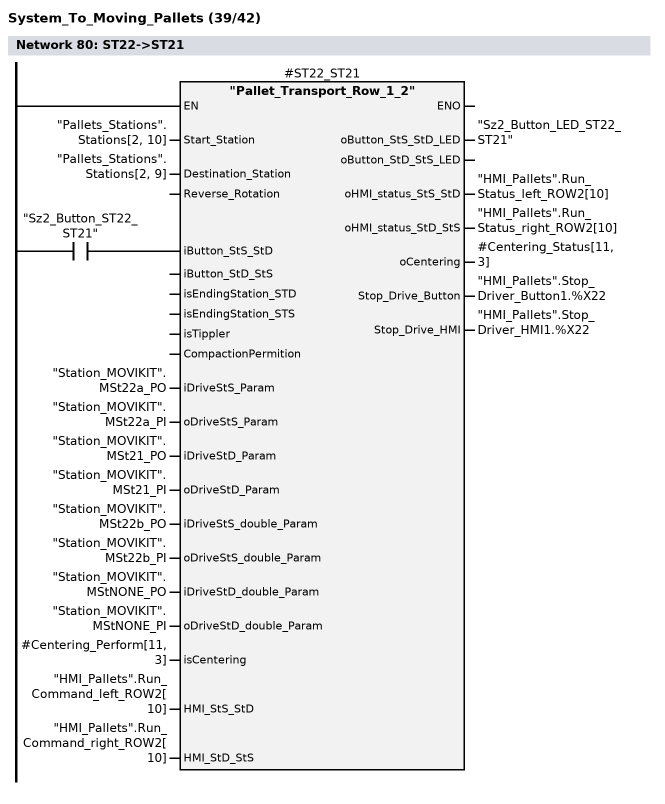
   RUNG wire#powerrail
      #ST22_ST21(iButton_StS_StD := wire#w1, Start_Station := "Pallets_Stations".Stations[2, 10], Destination_Station := "Pallets_Stations".Stations[2, 9], Reverse_Rotation :=, iButton_StD_StS :=, isEndingStation_STD :=, isEndingStation_STS :=, isTippler :=, CompactionPermition :=, iDriveStS_Param := "Station_MOVIKIT".MSt22a_PO, oDriveStS_Param := "Station_MOVIKIT".MSt22a_PI, iDriveStD_Param := "Station_MOVIKIT".MSt21_PO, oDriveStD_Param := "Station_MOVIKIT".MSt21_PI, iDriveStS_double_Param := "Station_MOVIKIT".MSt22b_PO, oDriveStS_double_Param := "Station_MOVIKIT".MSt22b_PI, iDriveStD_double_Param := "Station_MOVIKIT".MStNONE_PO, oDriveStD_double_Param := "Station_MOVIKIT".MStNONE_PI, isCentering := #Centering_Perform[11, 3], HMI_StS_StD := "HMI_Pallets".Run_Command_left_ROW2[10], HMI_StD_StS := "HMI_Pallets".Run_Command_right_ROW2[10], oButton_StS_StD_LED => "Sz2_Button_LED_ST22_ST21", oButton_StD_StS_LED =>, oHMI_status_StS_StD => "HMI_Pallets".Run_Status_left_ROW2[10], oHMI_status_StD_StS => "HMI_Pallets".Run_Status_right_ROW2[10], oCentering => #Centering_Status[11, 3], Stop_Drive_Button => "HMI_Pallets".Stop_Driver_Button1.%X22, Stop_Drive_HMI => "HMI_Pallets".Stop_Driver_HMI1.%X22)
   END_RUNG
   RUNG wire#powerrail
      Contact( "Sz2_Button_ST22_ST21" )
   END_RUNG wire#w1
   // the same network as SCL:
   #ST22_ST21(Start_Station := "Pallets_Stations".Stations[2, 10],   // "Pallet_Transport_Row_1_2"
              Destination_Station := "Pallets_Stations".Stations[2, 9],
              iButton_StS_StD := "Sz2_Button_ST22_ST21",
              iDriveStS_Param := "Station_MOVIKIT".MSt22a_PO,
              oDriveStS_Param := "Station_MOVIKIT".MSt22a_PI,
              iDriveStD_Param := "Station_MOVIKIT".MSt21_PO,
              oDriveStD_Param := "Station_MOVIKIT".MSt21_PI,
              iDriveStS_double_Param := "Station_MOVIKIT".MSt22b_PO,
              oDriveStS_double_Param := "Station_MOVIKIT".MSt22b_PI,
              iDriveStD_double_Param := "Station_MOVIKIT".MStNONE_PO,
              oDriveStD_double_Param := "Station_MOVIKIT".MStNONE_PI,
              isCentering := #Centering_Perform[11, 3],
              HMI_StS_StD := "HMI_Pallets".Run_Command_left_ROW2[10],
              HMI_StD_StS := "HMI_Pallets".Run_Command_right_ROW2[10],
              oButton_StS_StD_LED => "Sz2_Button_LED_ST22_ST21",
              oHMI_status_StS_StD => "HMI_Pallets".Run_Status_left_ROW2[10],
              oHMI_status_StD_StS => "HMI_Pallets".Run_Status_right_ROW2[10],
              oCentering => #Centering_Status[11, 3],
              Stop_Drive_Button => "HMI_Pallets".Stop_Driver_Button1.%X22,
              Stop_Drive_HMI => "HMI_Pallets".Stop_Driver_HMI1.%X22);
END_REGION

REGION Network 81: ST23->ST22
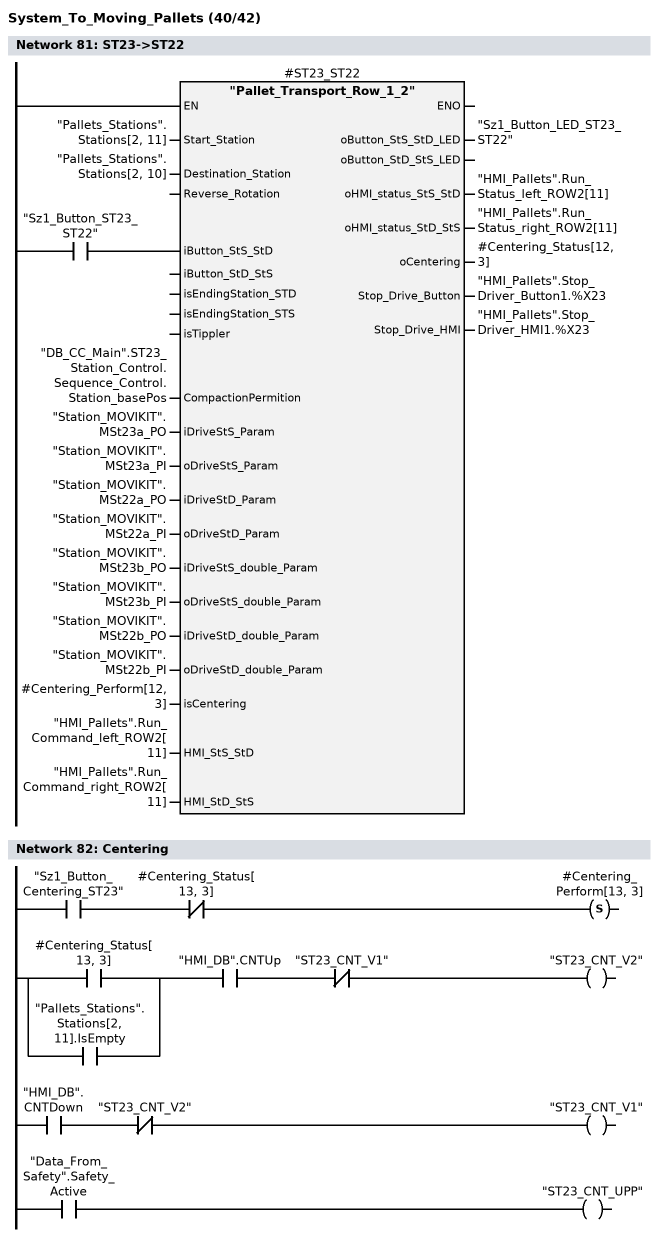
   RUNG wire#powerrail
      #ST23_ST22(iButton_StS_StD := wire#w1, Start_Station := "Pallets_Stations".Stations[2, 11], Destination_Station := "Pallets_Stations".Stations[2, 10], Reverse_Rotation :=, iButton_StD_StS :=, isEndingStation_STD :=, isEndingStation_STS :=, isTippler :=, CompactionPermition := "DB_CC_Main".ST23_Station_Control.Sequence_Control.Station_basePos, iDriveStS_Param := "Station_MOVIKIT".MSt23a_PO, oDriveStS_Param := "Station_MOVIKIT".MSt23a_PI, iDriveStD_Param := "Station_MOVIKIT".MSt22a_PO, oDriveStD_Param := "Station_MOVIKIT".MSt22a_PI, iDriveStS_double_Param := "Station_MOVIKIT".MSt23b_PO, oDriveStS_double_Param := "Station_MOVIKIT".MSt23b_PI, iDriveStD_double_Param := "Station_MOVIKIT".MSt22b_PO, oDriveStD_double_Param := "Station_MOVIKIT".MSt22b_PI, isCentering := #Centering_Perform[12, 3], HMI_StS_StD := "HMI_Pallets".Run_Command_left_ROW2[11], HMI_StD_StS := "HMI_Pallets".Run_Command_right_ROW2[11], oButton_StS_StD_LED => "Sz1_Button_LED_ST23_ST22", oButton_StD_StS_LED =>, oHMI_status_StS_StD => "HMI_Pallets".Run_Status_left_ROW2[11], oHMI_status_StD_StS => "HMI_Pallets".Run_Status_right_ROW2[11], oCentering => #Centering_Status[12, 3], Stop_Drive_Button => "HMI_Pallets".Stop_Driver_Button1.%X23, Stop_Drive_HMI => "HMI_Pallets".Stop_Driver_HMI1.%X23)
   END_RUNG
   RUNG wire#powerrail
      Contact( "Sz1_Button_ST23_ST22" )
   END_RUNG wire#w1
   // the same network as SCL:
   #ST23_ST22(Start_Station := "Pallets_Stations".Stations[2, 11],   // "Pallet_Transport_Row_1_2"
              Destination_Station := "Pallets_Stations".Stations[2, 10],
              iButton_StS_StD := "Sz1_Button_ST23_ST22",
              CompactionPermition := "DB_CC_Main".ST23_Station_Control.Sequence_Control.Station_basePos,
              iDriveStS_Param := "Station_MOVIKIT".MSt23a_PO,
              oDriveStS_Param := "Station_MOVIKIT".MSt23a_PI,
              iDriveStD_Param := "Station_MOVIKIT".MSt22a_PO,
              oDriveStD_Param := "Station_MOVIKIT".MSt22a_PI,
              iDriveStS_double_Param := "Station_MOVIKIT".MSt23b_PO,
              oDriveStS_double_Param := "Station_MOVIKIT".MSt23b_PI,
              iDriveStD_double_Param := "Station_MOVIKIT".MSt22b_PO,
              oDriveStD_double_Param := "Station_MOVIKIT".MSt22b_PI,
              isCentering := #Centering_Perform[12, 3],
              HMI_StS_StD := "HMI_Pallets".Run_Command_left_ROW2[11],
              HMI_StD_StS := "HMI_Pallets".Run_Command_right_ROW2[11],
              oButton_StS_StD_LED => "Sz1_Button_LED_ST23_ST22",
              oHMI_status_StS_StD => "HMI_Pallets".Run_Status_left_ROW2[11],
              oHMI_status_StD_StS => "HMI_Pallets".Run_Status_right_ROW2[11],
              oCentering => #Centering_Status[12, 3],
              Stop_Drive_Button => "HMI_Pallets".Stop_Driver_Button1.%X23,
              Stop_Drive_HMI => "HMI_Pallets".Stop_Driver_HMI1.%X23);
END_REGION

REGION Network 82: Centering
   RUNG wire#powerrail
      Contact( "Sz1_Button_Centering_ST23" )
      I_Contact( #Centering_Status[13, 3] )
      S_Coil( #Centering_Perform[13, 3] )
   END_RUNG
   RUNG wire#powerrail
      Contact( #Centering_Status[13, 3] )
      wire#w1
      Contact( "HMI_DB".CNTUp )
      I_Contact( "ST23_CNT_V1" )
      Coil( "ST23_CNT_V2" )
   END_RUNG
   RUNG wire#powerrail
      Contact( "Pallets_Stations".Stations[2, 11].IsEmpty )
   END_RUNG wire#w1
   RUNG wire#powerrail
      Contact( "HMI_DB".CNTDown )
      I_Contact( "ST23_CNT_V2" )
      Coil( "ST23_CNT_V1" )
   END_RUNG
   RUNG wire#powerrail
      Contact( "Data_From_Safety".Safety_Active )
      Coil( "ST23_CNT_UPP" )
   END_RUNG
   // the same network as SCL:
   IF "Sz1_Button_Centering_ST23" AND NOT #Centering_Status[13, 3] THEN
       #Centering_Perform[13, 3] := TRUE;
   END_IF;
   "ST23_CNT_V2" := (#Centering_Status[13, 3] OR "Pallets_Stations".Stations[2, 11].IsEmpty) AND "HMI_DB".CNTUp AND NOT "ST23_CNT_V1";
   "ST23_CNT_V1" := "HMI_DB".CNTDown AND NOT "ST23_CNT_V2";
   "ST23_CNT_UPP" := "Data_From_Safety".Safety_Active;
END_REGION

REGION Network 83: ST24->ST23
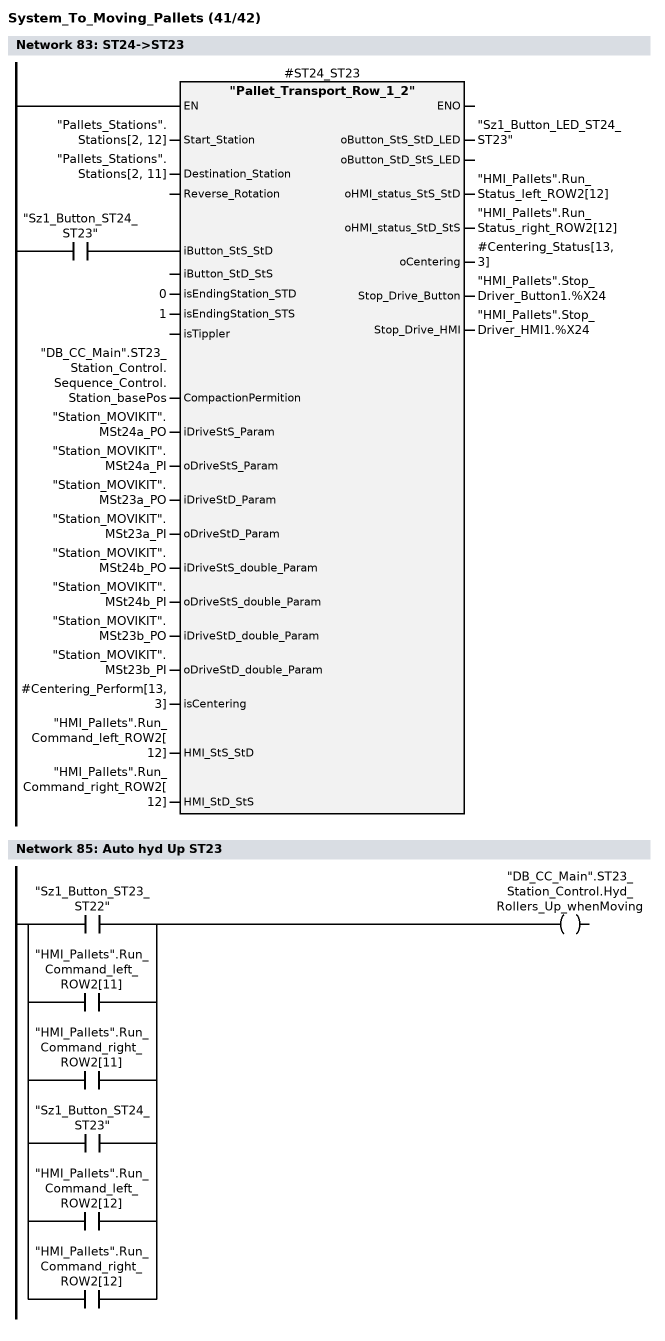
   RUNG wire#powerrail
      #ST24_ST23(iButton_StS_StD := wire#w1, Start_Station := "Pallets_Stations".Stations[2, 12], Destination_Station := "Pallets_Stations".Stations[2, 11], Reverse_Rotation :=, iButton_StD_StS :=, isEndingStation_STD := 0, isEndingStation_STS := 1, isTippler :=, CompactionPermition := "DB_CC_Main".ST23_Station_Control.Sequence_Control.Station_basePos, iDriveStS_Param := "Station_MOVIKIT".MSt24a_PO, oDriveStS_Param := "Station_MOVIKIT".MSt24a_PI, iDriveStD_Param := "Station_MOVIKIT".MSt23a_PO, oDriveStD_Param := "Station_MOVIKIT".MSt23a_PI, iDriveStS_double_Param := "Station_MOVIKIT".MSt24b_PO, oDriveStS_double_Param := "Station_MOVIKIT".MSt24b_PI, iDriveStD_double_Param := "Station_MOVIKIT".MSt23b_PO, oDriveStD_double_Param := "Station_MOVIKIT".MSt23b_PI, isCentering := #Centering_Perform[13, 3], HMI_StS_StD := "HMI_Pallets".Run_Command_left_ROW2[12], HMI_StD_StS := "HMI_Pallets".Run_Command_right_ROW2[12], oButton_StS_StD_LED => "Sz1_Button_LED_ST24_ST23", oButton_StD_StS_LED =>, oHMI_status_StS_StD => "HMI_Pallets".Run_Status_left_ROW2[12], oHMI_status_StD_StS => "HMI_Pallets".Run_Status_right_ROW2[12], oCentering => #Centering_Status[13, 3], Stop_Drive_Button => "HMI_Pallets".Stop_Driver_Button1.%X24, Stop_Drive_HMI => "HMI_Pallets".Stop_Driver_HMI1.%X24)
   END_RUNG
   RUNG wire#powerrail
      Contact( "Sz1_Button_ST24_ST23" )
   END_RUNG wire#w1
   // the same network as SCL:
   #ST24_ST23(Start_Station := "Pallets_Stations".Stations[2, 12],   // "Pallet_Transport_Row_1_2"
              Destination_Station := "Pallets_Stations".Stations[2, 11],
              iButton_StS_StD := "Sz1_Button_ST24_ST23",
              isEndingStation_STD := 0,
              isEndingStation_STS := 1,
              CompactionPermition := "DB_CC_Main".ST23_Station_Control.Sequence_Control.Station_basePos,
              iDriveStS_Param := "Station_MOVIKIT".MSt24a_PO,
              oDriveStS_Param := "Station_MOVIKIT".MSt24a_PI,
              iDriveStD_Param := "Station_MOVIKIT".MSt23a_PO,
              oDriveStD_Param := "Station_MOVIKIT".MSt23a_PI,
              iDriveStS_double_Param := "Station_MOVIKIT".MSt24b_PO,
              oDriveStS_double_Param := "Station_MOVIKIT".MSt24b_PI,
              iDriveStD_double_Param := "Station_MOVIKIT".MSt23b_PO,
              oDriveStD_double_Param := "Station_MOVIKIT".MSt23b_PI,
              isCentering := #Centering_Perform[13, 3],
              HMI_StS_StD := "HMI_Pallets".Run_Command_left_ROW2[12],
              HMI_StD_StS := "HMI_Pallets".Run_Command_right_ROW2[12],
              oButton_StS_StD_LED => "Sz1_Button_LED_ST24_ST23",
              oHMI_status_StS_StD => "HMI_Pallets".Run_Status_left_ROW2[12],
              oHMI_status_StD_StS => "HMI_Pallets".Run_Status_right_ROW2[12],
              oCentering => #Centering_Status[13, 3],
              Stop_Drive_Button => "HMI_Pallets".Stop_Driver_Button1.%X24,
              Stop_Drive_HMI => "HMI_Pallets".Stop_Driver_HMI1.%X24);
END_REGION

REGION Network 84 (SCL): Reset centering status of Tippler
   IF ("Station_MOVIKIT".MSt1_PO.x_Bit_1_Enable_Application_Stop OR "Station_MOVIKIT".MSt1a_PO.x_Bit_1_Enable_Application_Stop) AND #oCeterTippler THEN
       #Reset_Centering_Tippler := 1;
   ELSE
       #Reset_Centering_Tippler := 0;
   END_IF;
END_REGION

REGION Network 85: Auto hyd Up ST23
   RUNG wire#powerrail
      Contact( "Sz1_Button_ST23_ST22" )
      wire#w1
      Coil( "DB_CC_Main".ST23_Station_Control.Hyd_Rollers_Up_whenMoving )
   END_RUNG
   RUNG wire#powerrail
      Contact( "HMI_Pallets".Run_Command_left_ROW2[11] )
   END_RUNG wire#w1
   RUNG wire#powerrail
      Contact( "HMI_Pallets".Run_Command_right_ROW2[11] )
   END_RUNG wire#w1
   RUNG wire#powerrail
      Contact( "Sz1_Button_ST24_ST23" )
   END_RUNG wire#w1
   RUNG wire#powerrail
      Contact( "HMI_Pallets".Run_Command_left_ROW2[12] )
   END_RUNG wire#w1
   RUNG wire#powerrail
      Contact( "HMI_Pallets".Run_Command_right_ROW2[12] )
   END_RUNG wire#w1
   // the same network as SCL:
   "DB_CC_Main".ST23_Station_Control.Hyd_Rollers_Up_whenMoving := "Sz1_Button_ST23_ST22" OR "HMI_Pallets".Run_Command_left_ROW2[11] OR "HMI_Pallets".Run_Command_right_ROW2[11] OR "Sz1_Button_ST24_ST23" OR "HMI_Pallets".Run_Command_left_ROW2[12] OR "HMI_Pallets".Run_Command_right_ROW2[12];
END_REGION

REGION Network 86: Auto hyd Up ST24
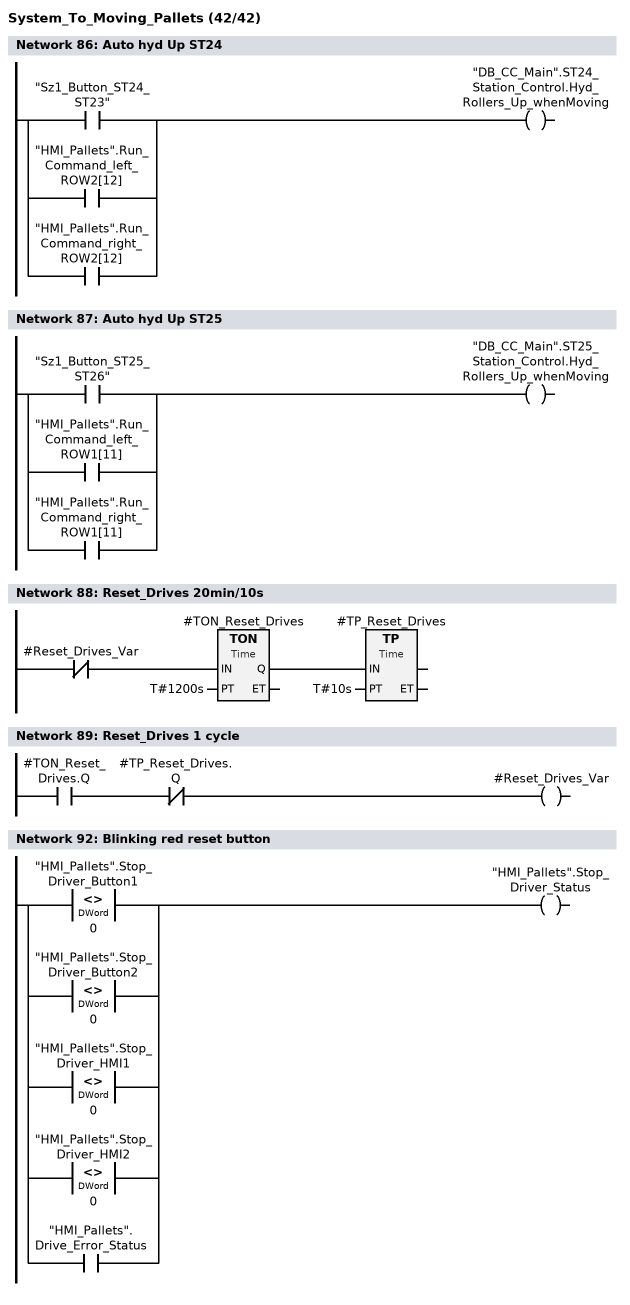
   RUNG wire#powerrail
      Contact( "Sz1_Button_ST24_ST23" )
      wire#w1
      Coil( "DB_CC_Main".ST24_Station_Control.Hyd_Rollers_Up_whenMoving )
   END_RUNG
   RUNG wire#powerrail
      Contact( "HMI_Pallets".Run_Command_left_ROW2[12] )
   END_RUNG wire#w1
   RUNG wire#powerrail
      Contact( "HMI_Pallets".Run_Command_right_ROW2[12] )
   END_RUNG wire#w1
   // the same network as SCL:
   "DB_CC_Main".ST24_Station_Control.Hyd_Rollers_Up_whenMoving := "Sz1_Button_ST24_ST23" OR "HMI_Pallets".Run_Command_left_ROW2[12] OR "HMI_Pallets".Run_Command_right_ROW2[12];
END_REGION

REGION Network 87: Auto hyd Up ST25
   RUNG wire#powerrail
      Contact( "Sz1_Button_ST25_ST26" )
      wire#w1
      Coil( "DB_CC_Main".ST25_Station_Control.Hyd_Rollers_Up_whenMoving )
   END_RUNG
   RUNG wire#powerrail
      Contact( "HMI_Pallets".Run_Command_left_ROW1[11] )
   END_RUNG wire#w1
   RUNG wire#powerrail
      Contact( "HMI_Pallets".Run_Command_right_ROW1[11] )
   END_RUNG wire#w1
   // the same network as SCL:
   "DB_CC_Main".ST25_Station_Control.Hyd_Rollers_Up_whenMoving := "Sz1_Button_ST25_ST26" OR "HMI_Pallets".Run_Command_left_ROW1[11] OR "HMI_Pallets".Run_Command_right_ROW1[11];
END_REGION

REGION Network 88: Reset_Drives 20min/10s
   RUNG wire#powerrail
      I_Contact( #Reset_Drives_Var )
      { S7_Templates := "time_type := Time" } #TON_Reset_Drives.TON(pt := T#1200s, et =>)
      { S7_Templates := "time_type := Time" } #TP_Reset_Drives.TP(pt := T#10s, et =>)
   END_RUNG
   // the same network as SCL:
   #TON_Reset_Drives(IN := NOT #Reset_Drives_Var, PT := T#1200s);   // TON
   #TP_Reset_Drives(IN := #TON_Reset_Drives.Q, PT := T#10s);   // TP
END_REGION

REGION Network 89: Reset_Drives 1 cycle
   RUNG wire#powerrail
      Contact( #TON_Reset_Drives.Q )
      I_Contact( #TP_Reset_Drives.Q )
      Coil( #Reset_Drives_Var )
   END_RUNG
   // the same network as SCL:
   #Reset_Drives_Var := #TON_Reset_Drives.Q AND NOT #TP_Reset_Drives.Q;
END_REGION

REGION Network 90 (SCL): Select Pallet
   FOR #i := 1 TO 24 DO
       IF #i = "HMI_Pallets".Number_Of_Pallet THEN
           "Pallets_Stations".Pallets[#i].IsSelected := 1;
       ELSE
           "Pallets_Stations".Pallets[#i].IsSelected := 0;
       END_IF;
   END_FOR;
END_REGION

REGION Network 91 (SCL): Cyclic reset drive command
   IF #Reset_Drives_Var THEN

       FOR #i := 1 TO 12 DO
           "HMI_Pallets".Run_Command_left_ROW1[#i] := FALSE;
           "HMI_Pallets".Run_Command_left_ROW2[#i] := FALSE;
           "HMI_Pallets".Run_Command_left_ROW4[#i] := FALSE;
           "HMI_Pallets".Run_Command_right_ROW1[#i] := FALSE;
           "HMI_Pallets".Run_Command_right_ROW2[#i] := FALSE;
           "HMI_Pallets".Run_Command_right_ROW4[#i] := FALSE;
       END_FOR;
   END_IF;
END_REGION

REGION Network 92: Blinking red reset button
   RUNG wire#powerrail
      { S7_Templates := "SrcType := DWord" } NE_Contact(in1 := "HMI_Pallets".Stop_Driver_Button1, in2 := 0)
      wire#w1
      Coil( "HMI_Pallets".Stop_Driver_Status )
   END_RUNG
   RUNG wire#powerrail
      { S7_Templates := "SrcType := DWord" } NE_Contact(in1 := "HMI_Pallets".Stop_Driver_Button2, in2 := 0)
   END_RUNG wire#w1
   RUNG wire#powerrail
      { S7_Templates := "SrcType := DWord" } NE_Contact(in1 := "HMI_Pallets".Stop_Driver_HMI1, in2 := 0)
   END_RUNG wire#w1
   RUNG wire#powerrail
      { S7_Templates := "SrcType := DWord" } NE_Contact(in1 := "HMI_Pallets".Stop_Driver_HMI2, in2 := 0)
   END_RUNG wire#w1
   RUNG wire#powerrail
      Contact( "HMI_Pallets".Drive_Error_Status )
   END_RUNG wire#w1
   // the same network as SCL:
   "HMI_Pallets".Stop_Driver_Status := ("HMI_Pallets".Stop_Driver_Button1 <> 0) OR ("HMI_Pallets".Stop_Driver_Button2 <> 0) OR ("HMI_Pallets".Stop_Driver_HMI1 <> 0) OR ("HMI_Pallets".Stop_Driver_HMI2 <> 0) OR "HMI_Pallets".Drive_Error_Status;
END_REGION

REGION Network 93 (SCL)
   REGION W1 Reset
       // Timer ON when Command_Run_W1 = 1
       #tComm_W1(IN := "HMI_Pallets".Command_Run_W1,
                 PT := T#2m);

       // Reset after 2m
       IF #tComm_W1.Q THEN
           "HMI_Pallets".Command_Run_W1 := FALSE;
       END_IF;

   END_REGION

   REGION W2 Reset
       // Timer ON when Command_Run_W2 = 1
       #tComm_W2(IN := "HMI_Pallets".Command_Run_W2,
                 PT := T#2m);

       // Reset after 2m
       IF #tComm_W2.Q THEN
           "HMI_Pallets".Command_Run_W2 := FALSE;
       END_IF;

   END_REGION


   REGION W4 Reset
       // Timer ON when Command_Run_W4 = 1
       #tComm_W4(IN := "HMI_Pallets".Command_Run_W4,
                 PT := T#2m);

       // Reset after 2m
       IF #tComm_W4.Q THEN
           "HMI_Pallets".Command_Run_W4 := FALSE;
       END_IF;

   END_REGION

   //TO DO change W1 & W2 to W1_2 
   IF (
       ("HMI_Pallets".Command_Run_W1 AND "HMI_Pallets".Command_Run_W2) OR
       ("HMI_Pallets".Command_Run_W1 AND "HMI_Pallets".Command_Run_W4) OR
       ("HMI_Pallets".Command_Run_W2 AND "HMI_Pallets".Command_Run_W4)
       ) THEN

       "HMI_Pallets".Command_Run_W1 := FALSE;
       "HMI_Pallets".Command_Run_W2 := FALSE;
       "HMI_Pallets".Command_Run_W4 := FALSE;

   END_IF;
END_REGION
END_FUNCTION_BLOCK
